(* IEC 61131-3 sources: PneuTrunk/pneutrunk_plc/Source/UDP/Server, 2 files *)

(* ---- Server.st ---- *)
(********************************************************************
 * COPYRIGHT -- Bernecker + Rainer
 ********************************************************************
 * Program: Server
 * File: Server.st
 * Author: Bernecker + Rainer
 * Created: June 02, 2008
 ********************************************************************
 * Implementation of program Server
 ********************************************************************)

PROGRAM _CYCLIC

	CASE Server.sStep OF

		0:	(* Open UDP Port *)
			Server.UdpOpen_0.enable := 1;
			Server.UdpOpen_0.pIfAddr := 0;	(* Listen on all TCP/IP Interfaces*)
			Server.UdpOpen_0.port := 12050;	(* Port to listen*)
			Server.UdpOpen_0.options := 0;
			Server.UdpOpen_0;	(* Call the Function*)

			IF Server.UdpOpen_0.status = 0 THEN  (* UdpOpen successful*)
				Server.sStep := 1;
			ELSIF Server.UdpOpen_0.status = ERR_FUB_BUSY THEN  (* UdpOpen not finished -> redo *)
			  (* Busy *)
			ELSE  (* Goto Error Step *)
				Server.sStep := 10;
			END_IF

		1:	(* Wait for Data *)
			Server.UdpRecv_0.enable := 1;
			Server.UdpRecv_0.ident := Server.UdpOpen_0.ident;	(* Client Ident from AsUDP.UDP_Open *)
			Server.UdpRecv_0.pData := ADR(Server.data_buffer);	(* Where to store the incoming data *)
			Server.UdpRecv_0.datamax := SIZEOF(Server.data_buffer);	(* Lenght of data buffer *)
			Server.UdpRecv_0.flags := 0;
			Server.UdpRecv_0.pIpAddr := ADR(Server.client_address);	(* IP Address of the Client *)
			Server.UdpRecv_0;	(* Call the Function*)

			IF Server.UdpRecv_0.status = 0 THEN  (* Data received *)
				Server.sStep := 2;
			ELSIF Server.UdpRecv_0.status = udpERR_NO_DATA THEN  (* No data received - wait *)
			  (* No Data received *)
			ELSIF Server.UdpRecv_0.status = ERR_FUB_BUSY THEN  (* UdpRecv not finished -> redo *)
			  (* Busy *)
			ELSE  (* Goto Error Step *)
				Server.sStep := 10;
			END_IF

		2:	(* Send Data back to Client *)

			Server.UdpSend_0.enable := 1;
			Server.UdpSend_0.ident := Server.UdpOpen_0.ident;	// Client Ident from AsUDP.UDP_Open
			Server.UdpSend_0.pHost := ADR(Server.client_address);	// IP Address of the Client
			Server.UdpSend_0.port := Server.UdpRecv_0.port;		// Port number of the Client
			Server.UdpSend_0.pData := ADR(Server.data_buffer);	// Which data to send
			Server.UdpSend_0.datalen := SIZEOF(Server.data_buffer);	// Lenght of data to send
			Server.UdpSend_0.flags := 0;
			Server.UdpSend_0;	// Call the Function

			IF switch = FALSE THEN
				// Yellow - 1, Red - 2, Undefined - 3
				packetPos.color := FIND(Server.data_buffer, 'yellow');
				IF(packetPos.color>1)THEN
					automatika.step_color := 1;
				ELSIF(packetPos.color=0)THEN
					packetPos.color := FIND(Server.data_buffer, 'red');
					IF(packetPos.color>1) THEN
						automatika.step_color:= 2;
					ELSE
						automatika.step_color:= 3;
					END_IF

				END_IF
				// Volba kroku robota
				packetPos.step := FIND(Server.data_buffer, 'come');
				IF(packetPos.step >1)THEN
					global_step_udp := 1;
				ELSIF(packetPos.step = 0)THEN
					packetPos.step := FIND(Server.data_buffer, 'hold');
					IF(packetPos.step >1)THEN
						global_step_udp := 2;
					ELSIF(packetPos.step = 0)THEN
						packetPos.step := FIND(Server.data_buffer, 'release');
						IF(packetPos.step >1)THEN
							global_step_udp := 3;
						ELSIF(packetPos.step = 0)THEN
							packetPos.step := FIND(Server.data_buffer, 'continue');
							IF(packetPos.step >1)THEN
								global_step_udp := 4;
							END_IF
						END_IF
					END_IF
				END_IF

				packetPos.q := FIND(Server.data_buffer, 'q:');
				packetPos.c := FIND(Server.data_buffer, 'c:'); // Server.data_buffer bolo povodne ked to slo STRING[5][0..100] a tu bolo Server.data_buffer[0]
				packetPos.qLength := UDINT_TO_INT(Server.UdpSend_0.datalen) - (packetPos.q + 1) - packetPos.c;
				packetPos.qFull := MID(Server.data_buffer, packetPos.c-packetPos.q-2, packetPos.q+2);
				FOR i:=0 TO 13 BY 1 DO	//11
					packetPos.comma := FIND(packetPos.qFull, ',');
					packetPos.qString[i] := MID(packetPos.qFull, packetPos.comma, 0);
					packetPos.qFull := DELETE(packetPos.qFull, packetPos.comma+1, 0);
					packetPos.qDesired[i] := atof(ADR(packetPos.qString[i])) ;
				END_FOR
				packetPos.qString[14] := MID(packetPos.qFull, packetPos.comma, 0);//12
				packetPos.qFull := DELETE(packetPos.qFull, packetPos.comma+1, 0);
				packetPos.qDesired[14] := atof(ADR(packetPos.qString[14]));//12
			END_IF

			IF Server.UdpSend_0.status = 0 THEN  (* Data sent *)
				Server.sStep := 1;
			ELSIF Server.UdpSend_0.status = ERR_FUB_BUSY THEN  (* UdpSend not finished -> redo *)
			  (* Busy *)
			ELSE  (* Goto Error Step *)
				Server.sStep := 10;
			END_IF

		10:  (* Here some error Handling has to be implemented *)

	END_CASE

END_PROGRAM

(* ---- Server.var ---- *)
(********************************************************************
 * COPYRIGHT -- Bernecker + Rainer
 ********************************************************************
 * Program: Server
 * File: Server.var
 * Author: Bernecker + Rainer
 * Created: June 02, 2008
 ********************************************************************
 * Local variables of program Server
 ********************************************************************)
VAR
	Server : Server_typ := (0); (*Data for Server Task*)
	i : INT;
	switch : BOOL;
END_VAR
